# EPICS substitutions: db/ecmcEL9505.substitutions
file ecmcEcSlave.template
{
    pattern {}
            {}
}

file ecmcEL9505.template
{
	pattern {}
		    {}
}
